// TIA Portal V14 export
DATA_BLOCK "DB_Outputs"   // DB1
// stored: AutoNumber true
BEGIN
END_DATA_BLOCK
